TYPE Beckhoff_AI :
STRUCT
	rawValue : WORD;
	OutOfRange : BOOL;
	Offline : BOOL;
	Value : REAL;
	
END_STRUCT
END_TYPE

(* stored: Version 1.1.0.1, ProductVersion 3.1.4024.12
   DUT Beckhoff_AI: Id {8c02a941-77e2-4143-9722-ae3fb28e6b49} *)
